% RSLogix 500 project PROJECT 1 CGT PART 4.RSS, saved by version 8.30.00.16 %
PROJECT "UNTITLED"    % processor: Bul.1763 MicroLogix 1100 Series B %

PROGRAM FILES
  LAD 2 "SECTIONS"  4 rungs
  LAD 3 "INPUT"  3 rungs
  LAD 4 "LOGIC"  8 rungs
  LAD 5 "OUTPUT"  4 rungs

DATA FILES
  O0 OUTPUT  4 elements
  I1 INPUT  6 elements
  S2 STATUS  66 elements
  B3 BINARY  1 elements
  T4 TIMER  2 elements
  C5 COUNTER  1 elements
  R6 CONTROL  1 elements
  N7 INTEGER  1 elements
  F8 FLOAT  1 elements

LADDER 2 "SECTIONS"
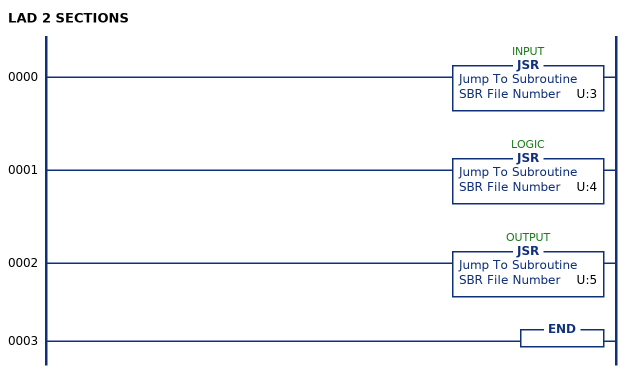
% Rung: 0 %
SOR JSR U:3 EOR
%   U:3  "INPUT" %
% Rung: 1 %
SOR JSR U:4 EOR
%   U:4  "LOGIC" %
% Rung: 2 %
SOR JSR U:5 EOR
%   U:5  "OUTPUT" %
% Rung: 3 %
SOR END EOR

LADDER 3 "INPUT"
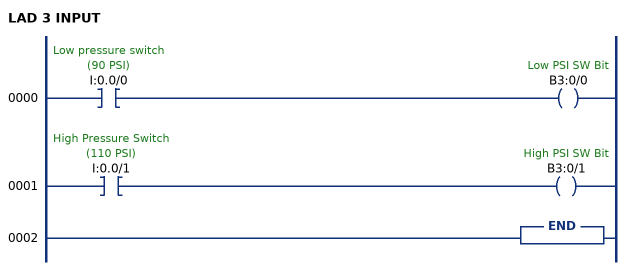
% Rung: 0 %
SOR XIC I:0.0/0 OTE B3:0/0 EOR
%   I:0.0/0  "Low pressure switch (90 PSI)" %
%   B3:0/0  "Low PSI SW Bit" %
% Rung: 1 %
SOR XIC I:0.0/1 OTE B3:0/1 EOR
%   I:0.0/1  "High Pressure Switch (110 PSI)" %
%   B3:0/1  "High PSI SW Bit" %
% Rung: 2 %
SOR END EOR

LADDER 4 "LOGIC"
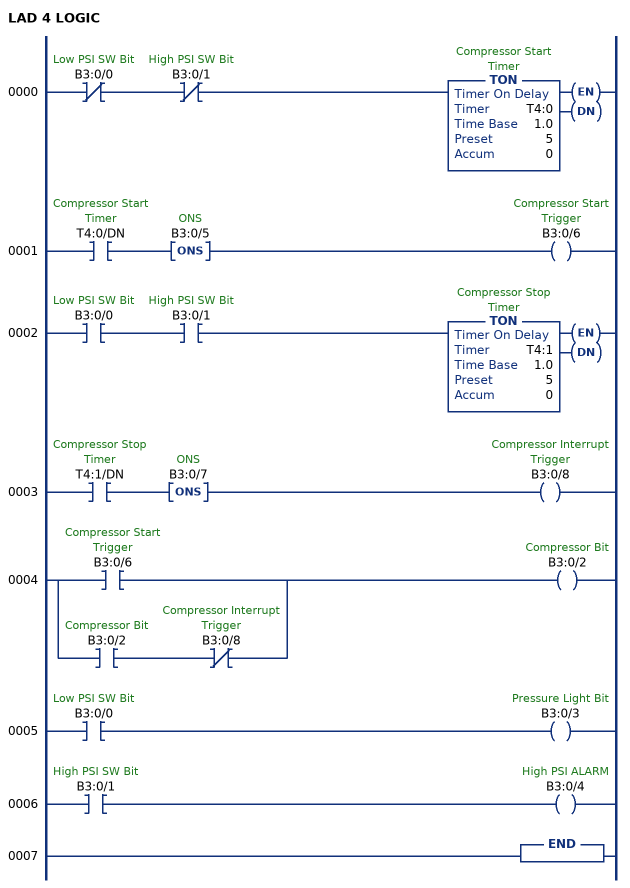
% Rung: 0 %
SOR XIO B3:0/0 XIO B3:0/1 TON T4:0 1.0 5 0 EOR
%   B3:0/0  "Low PSI SW Bit" %
%   B3:0/1  "High PSI SW Bit" %
%   T4:0  "Compressor Start Timer" %
% Rung: 1 %
SOR XIC T4:0/DN ONS B3:0/5 OTE B3:0/6 EOR
%   T4:0  "Compressor Start Timer" %
%   B3:0/5  "ONS" %
%   B3:0/6  "Compressor Start Trigger" %
% Rung: 2 %
SOR XIC B3:0/0 XIC B3:0/1 TON T4:1 1.0 5 0 EOR
%   B3:0/0  "Low PSI SW Bit" %
%   B3:0/1  "High PSI SW Bit" %
%   T4:1  "Compressor Stop Timer" %
% Rung: 3 %
SOR XIC T4:1/DN ONS B3:0/7 OTE B3:0/8 EOR
%   T4:1  "Compressor Stop Timer" %
%   B3:0/7  "ONS" %
%   B3:0/8  "Compressor Interrupt Trigger" %
% Rung: 4 %
SOR BST XIC B3:0/6 NXB XIC B3:0/2 XIO B3:0/8 BND OTE B3:0/2 EOR
%   B3:0/6  "Compressor Start Trigger" %
%   B3:0/2  "Compressor Bit" %
%   B3:0/8  "Compressor Interrupt Trigger" %
% Rung: 5 %
SOR XIC B3:0/0 OTE B3:0/3 EOR
%   B3:0/0  "Low PSI SW Bit" %
%   B3:0/3  "Pressure Light Bit" %
% Rung: 6 %
SOR XIC B3:0/1 OTE B3:0/4 EOR
%   B3:0/1  "High PSI SW Bit" %
%   B3:0/4  "High PSI ALARM" %
% Rung: 7 %
SOR END EOR

LADDER 5 "OUTPUT"
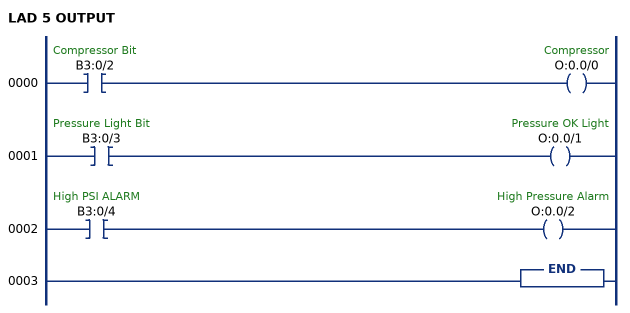
% Rung: 0 %
SOR XIC B3:0/2 OTE O:0.0/0 EOR
%   B3:0/2  "Compressor Bit" %
%   O:0.0/0  "Compressor" %
% Rung: 1 %
SOR XIC B3:0/3 OTE O:0.0/1 EOR
%   B3:0/3  "Pressure Light Bit" %
%   O:0.0/1  "Pressure OK Light" %
% Rung: 2 %
SOR XIC B3:0/4 OTE O:0.0/2 EOR
%   B3:0/4  "High PSI ALARM" %
%   O:0.0/2  "High Pressure Alarm" %
% Rung: 3 %
SOR END EOR

OTHER DOCUMENTED ADDRESSES
  T4:0/0  "Compressor Start Trigger"

DATA TABLE (non-zero values as saved)
DATA T4
% .PRE .ACC %
% T4:0 % 5 0
% T4:1 % 5 0
